# B&R Automation Studio project MOCS_AS
Automation Studio 4.12.5.95 SP

## Configuration GE3

CPU X20CP1686X, AutomationRuntime K4.93, Build 4.1.2, Vc V4.73.1

### Task classes (Cpu.sw)
```
Cyclic#4:
  IODiver <- IODefinitions.IODiver.prg
  CtrlLogic <- CtrlLogic.prg [disabled] (AdditionalIncludeDirectories=\Logical\MATLAB_includes\R2022b\, BuildOptions=-lm -DMODEL=MOCS_AS_Gen -DNUMST=1 -DNCSTATES=0 -DHAVESTDIO -DMODEL_HAS_DYNAMICALLY_LOADED_SFCNS=0 -DCLASSIC_INTERFACE=0 -DALLOCATIONFCN=0 -DTID01EQ=0 -DTERMFCN=1 -DONESTEPFCN=0 -DMAT_FILE=0 -DMULTI_INSTANCE_CODE=0 -DINTEGER_CODE=0 -DMT=0 )
Binaries: FWRules, udbdef, TCData, sysconf, asfw, User, iomap, arconfig, ashwd, Role, ashwac
Libraries: brsystem, asieccon, astime, runtime, sys_lib
```

### Hardware
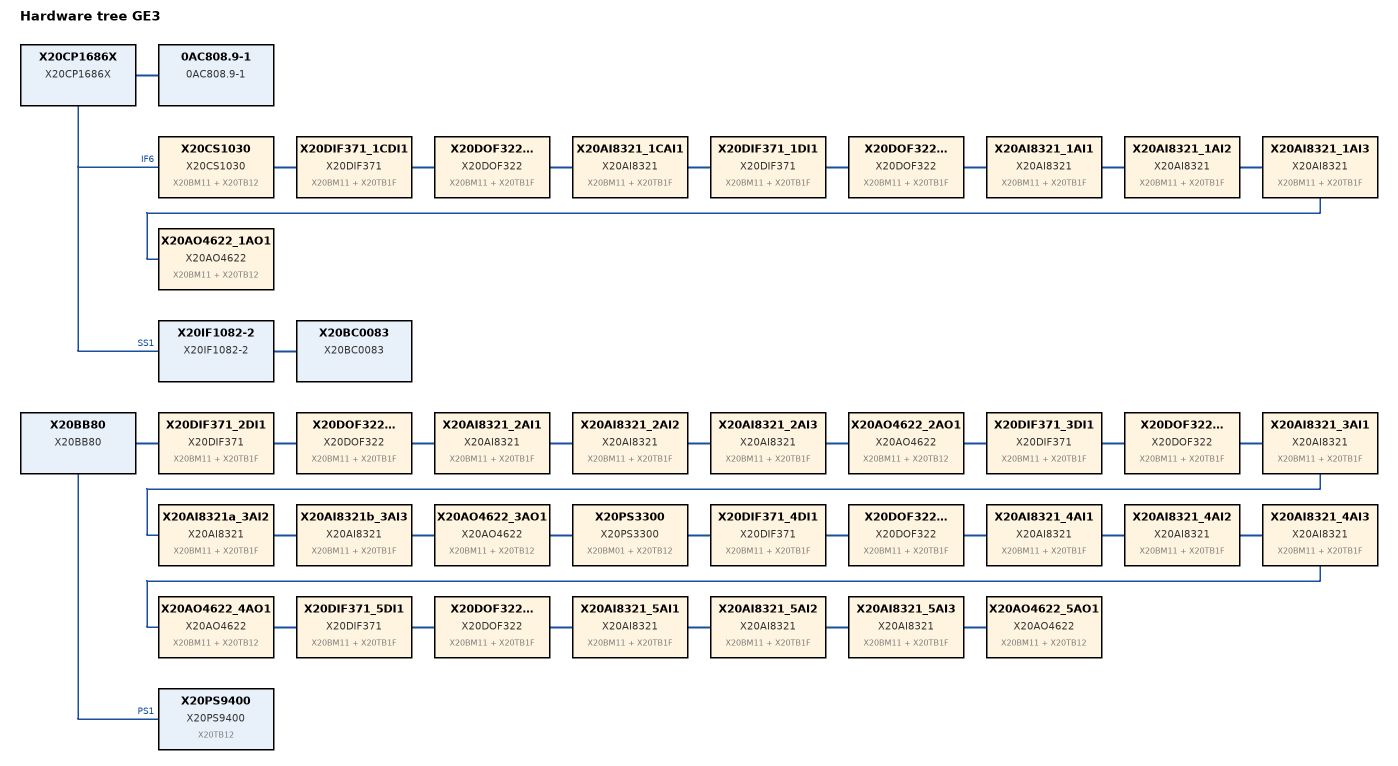
```
0AC808.9-1 : 0AC808.9-1 v1.0.0.0  [ETH1 -> X20CP1686X.IF2 [Cable Type=PowerlinkCable, Length=10, Version=1.0.0.3]]
X20AI8321_1AI1 : X20AI8321 v1.5.0.0  [SS1 -> X20TB1F5.SS; SL -> X20BM11f.SL1]
X20AI8321_1AI2 : X20AI8321 v1.5.0.0  [SS1 -> X20TB1F6.SS; SL -> X20BM11g.SL1]
X20AI8321_1AI3 : X20AI8321 v1.5.0.0  [SS1 -> X20TB1F7.SS; SL -> X20BM11h.SL1]
X20AI8321_1CAI1 : X20AI8321 v1.5.0.0  [SS1 -> X20TB1F2.SS; SL -> X20BM11c.SL1]
X20AI8321_2AI1 : X20AI8321 v1.5.0.0  [SS1 -> X20TB1F11.SS; SL -> X20BM11m.SL1]
X20AI8321_2AI2 : X20AI8321 v1.5.0.0  [SS1 -> X20TB1F12.SS; SL -> X20BM11n.SL1]
X20AI8321_2AI3 : X20AI8321 v1.5.0.0  [SS1 -> X20TB1F13.SS; SL -> X20BM11o.SL1]
X20AI8321_3AI1 : X20AI8321 v1.5.0.0  [SS1 -> X20TB1F15.SS; SL -> X20BM11r.SL1]
X20AI8321_4AI1 : X20AI8321 v1.5.0.0  [SS1 -> X20TB1F20.SS; SL -> X20BM11x.SL1]
X20AI8321_4AI2 : X20AI8321 v1.5.0.0  [SS1 -> X20TB1F21.SS; SL -> X20BM11y.SL1]
X20AI8321_4AI3 : X20AI8321 v1.5.0.0  [SS1 -> X20TB1F22.SS; SL -> X20BM11z.SL1]
X20AI8321_5AI1 : X20AI8321 v1.5.0.0  [SS1 -> X20TB1F25.SS; SL -> X20BM11ad.SL1]
X20AI8321_5AI2 : X20AI8321 v1.5.0.0  [SS1 -> X20TB1F26.SS; SL -> X20BM11ae.SL1]
X20AI8321_5AI3 : X20AI8321 v1.5.0.0  [SS1 -> X20TB1F27.SS; SL -> X20BM11af.SL1]
X20AI8321a_3AI2 : X20AI8321 v1.5.0.0  [SS1 -> X20TB1F16.SS; SL -> X20BM11s.SL1]
X20AI8321b_3AI3 : X20AI8321 v1.5.0.0  [SS1 -> X20TB1F17.SS; SL -> X20BM11t.SL1]
X20AO4622_1AO1 : X20AO4622 v1.4.1.0  [SS1 -> X20TB12a.SS; SL -> X20BM11i.SL1]
X20AO4622_2AO1 : X20AO4622 v1.4.1.0  [SS1 -> X20TB12c.SS; SL -> X20BM11l.SL1]
X20AO4622_3AO1 : X20AO4622 v1.4.1.0  [SS1 -> X20TB12d.SS; SL -> X20BM11u.SL1]
X20AO4622_4AO1 : X20AO4622 v1.4.1.0  [SS1 -> X20TB12e.SS; SL -> X20BM11aa.SL1]
X20AO4622_5AO1 : X20AO4622 v1.4.1.0  [SS1 -> X20TB12g.SS; SL -> X20BM11ag.SL1]
X20BB80 : X20BB80 v1.1.0.0
X20BC0083 : X20BC0083 v2.16.0.0  [PLK1 -> X20IF1082-2.IF1 (NodeNumber=1) [Cable Type=PowerlinkCable, Length=10, Version=1.0.0.3]; SL -> X20BB80.SL1]
X20BM01 : X20BM01 v2.2.0.0  [X2X1 -> X20BM11u.X2X2]
X20BM11 : X20BM11 v1.1.0.0  [X2X1 -> X20CP1686X.IF6]
X20BM11a : X20BM11 v1.1.0.0  [X2X1 -> X20BM11.X2X2]
X20BM11aa : X20BM11 v1.1.0.0  [X2X1 -> X20BM11z.X2X2]
X20BM11ab : X20BM11 v1.1.0.0  [X2X1 -> X20BM11aa.X2X2]
X20BM11ac : X20BM11 v1.1.0.0  [X2X1 -> X20BM11ab.X2X2]
X20BM11ad : X20BM11 v1.1.0.0  [X2X1 -> X20BM11ac.X2X2]
X20BM11ae : X20BM11 v1.1.0.0  [X2X1 -> X20BM11ad.X2X2]
X20BM11af : X20BM11 v1.1.0.0  [X2X1 -> X20BM11ae.X2X2]
X20BM11ag : X20BM11 v1.1.0.0  [X2X1 -> X20BM11af.X2X2]
X20BM11b : X20BM11 v1.1.0.0  [X2X1 -> X20BM11a.X2X2]
X20BM11c : X20BM11 v1.1.0.0  [X2X1 -> X20BM11b.X2X2]
X20BM11d : X20BM11 v1.1.0.0  [X2X1 -> X20BM11c.X2X2]
X20BM11e : X20BM11 v1.1.0.0  [X2X1 -> X20BM11d.X2X2]
X20BM11f : X20BM11 v1.1.0.0  [X2X1 -> X20BM11e.X2X2]
X20BM11g : X20BM11 v1.1.0.0  [X2X1 -> X20BM11f.X2X2]
X20BM11h : X20BM11 v1.1.0.0  [X2X1 -> X20BM11g.X2X2]
X20BM11i : X20BM11 v1.1.0.0  [X2X1 -> X20BM11h.X2X2]
X20BM11j : X20BM11 v1.1.0.0  [X2X1 -> X20BB80.IF1]
X20BM11k : X20BM11 v1.1.0.0  [X2X1 -> X20BM11j.X2X2]
X20BM11l : X20BM11 v1.1.0.0  [X2X1 -> X20BM11o.X2X2]
X20BM11m : X20BM11 v1.1.0.0  [X2X1 -> X20BM11k.X2X2]
X20BM11n : X20BM11 v1.1.0.0  [X2X1 -> X20BM11m.X2X2]
X20BM11o : X20BM11 v1.1.0.0  [X2X1 -> X20BM11n.X2X2]
X20BM11p : X20BM11 v1.1.0.0  [X2X1 -> X20BM11l.X2X2]
X20BM11q : X20BM11 v1.1.0.0  [X2X1 -> X20BM11p.X2X2]
X20BM11r : X20BM11 v1.1.0.0  [X2X1 -> X20BM11q.X2X2]
X20BM11s : X20BM11 v1.1.0.0  [X2X1 -> X20BM11r.X2X2]
X20BM11t : X20BM11 v1.1.0.0  [X2X1 -> X20BM11s.X2X2]
X20BM11u : X20BM11 v1.1.0.0  [X2X1 -> X20BM11t.X2X2]
X20BM11v : X20BM11 v1.1.0.0  [X2X1 -> X20BM01.X2X2]
X20BM11w : X20BM11 v1.1.0.0  [X2X1 -> X20BM11v.X2X2]
X20BM11x : X20BM11 v1.1.0.0  [X2X1 -> X20BM11w.X2X2]
X20BM11y : X20BM11 v1.1.0.0  [X2X1 -> X20BM11x.X2X2]
X20BM11z : X20BM11 v1.1.0.0  [X2X1 -> X20BM11y.X2X2]
X20CP1686X : X20CP1686X v1.6.2.0
  Connector IF2:
    ActivateDevice = 1
    HostName = multimocs
    Mode = Manual
    InternetAddress = 172.16.8.77
    SubnetMask = 255.255.255.0
  Connector IF3:
    EplHostName = multimocs
    HostName = multimocs
  ConfigurationID = MultiMOCS
  FileDevice1
  FileDeviceName1 = USER
  FileDevicePath1 = F:\
  FileDevice2
  FileDeviceName2 = USB_DEVICE
  FileDevicePath2 = /bd0
  FileDevice3
  FileDeviceName3 = ALARM_HISTROY
  FileDevicePath3 = F:\ALARM_HISTROY
  FileDevice4
  FileDeviceName4 = RECIPE
  FileDevicePath4 = F:\RECIPE
  FileDevice5
  FileDeviceName5 = AUDIT
  FileDevicePath5 = F:\AUDIT
  TimeZone = 325
  EthernetHostName = multimocs
  FtpUser1
  FtpUsername1 = hhi
  FtpUserPassword1 = NOQKJFEIpCMGTGhB1oqHL8VzUKYS3v77UCmMnhUHHNQ=
  FtpUserSalt1 = B7uzC8IW
  FTPAccessRight1 = 0
  ActivateOpcUa = 1
  OpcUaInformationModels_PV_Version = 1
X20CS1030 : X20CS1030 v1.8.0.0  [SS1 -> X20TB12.SS; SL -> X20BM11.SL1]
X20DIF371_1CDI1 : X20DIF371 v1.4.0.0  [SS1 -> X20TB1F.SS; SL -> X20BM11a.SL1]
X20DIF371_1DI1 : X20DIF371 v1.4.0.0  [SS1 -> X20TB1F3.SS; SL -> X20BM11d.SL1]
X20DIF371_2DI1 : X20DIF371 v1.4.0.0  [SS1 -> X20TB1F8.SS; SL -> X20BM11j.SL1]
X20DIF371_3DI1 : X20DIF371 v1.4.0.0  [SS1 -> X20TB1F10.SS; SL -> X20BM11p.SL1]
X20DIF371_4DI1 : X20DIF371 v1.4.0.0  [SS1 -> X20TB1F18.SS; SL -> X20BM11v.SL1]
X20DIF371_5DI1 : X20DIF371 v1.4.0.0  [SS1 -> X20TB1F23.SS; SL -> X20BM11ab.SL1]
X20DOF322_1CDO1 : X20DOF322 v1.5.0.0  [SS1 -> X20TB1F1.SS; SL -> X20BM11b.SL1]
X20DOF322_1DO1 : X20DOF322 v1.5.0.0  [SS1 -> X20TB1F4.SS; SL -> X20BM11e.SL1]
X20DOF322_2DO1 : X20DOF322 v1.5.0.0  [SS1 -> X20TB1F9.SS; SL -> X20BM11k.SL1]
X20DOF322_3DO1 : X20DOF322 v1.5.0.0  [SS1 -> X20TB1F14.SS; SL -> X20BM11q.SL1]
X20DOF322_4DO1 : X20DOF322 v1.5.0.0  [SS1 -> X20TB1F19.SS; SL -> X20BM11w.SL1]
X20DOF322_5DO1 : X20DOF322 v1.5.0.0  [SS1 -> X20TB1F24.SS; SL -> X20BM11ac.SL1]
X20IF1082-2 : X20IF1082-2 v1.15.0.0  [SS -> X20CP1686X.SS1]
  Connector IF1:
    EplHostName = multimocs
    EplNatSubnet = 192.168.102.0
    HostName = multimocs
X20PS3300 : X20PS3300 v1.4.0.0  [SS1 -> X20TB12f.SS; SL -> X20BM01.SL1]
X20PS9400 : X20PS9400 v1.8.0.0  [SS1 -> X20TB12b.SS; PS -> X20BB80.PS1]
X20TB12 : X20TB12 v1.0.0.0
X20TB12a : X20TB12 v1.0.0.0
X20TB12b : X20TB12 v1.0.0.0
X20TB12c : X20TB12 v1.0.0.0
X20TB12d : X20TB12 v1.0.0.0
X20TB12e : X20TB12 v1.0.0.0
X20TB12f : X20TB12 v1.0.0.0
X20TB12g : X20TB12 v1.0.0.0
X20TB1F : X20TB1F v1.0.0.0
X20TB1F1 : X20TB1F v1.0.0.0
X20TB1F10 : X20TB1F v1.0.0.0
X20TB1F11 : X20TB1F v1.0.0.0
X20TB1F12 : X20TB1F v1.0.0.0
X20TB1F13 : X20TB1F v1.0.0.0
X20TB1F14 : X20TB1F v1.0.0.0
X20TB1F15 : X20TB1F v1.0.0.0
X20TB1F16 : X20TB1F v1.0.0.0
X20TB1F17 : X20TB1F v1.0.0.0
X20TB1F18 : X20TB1F v1.0.0.0
X20TB1F19 : X20TB1F v1.0.0.0
X20TB1F2 : X20TB1F v1.0.0.0
X20TB1F20 : X20TB1F v1.0.0.0
X20TB1F21 : X20TB1F v1.0.0.0
X20TB1F22 : X20TB1F v1.0.0.0
X20TB1F23 : X20TB1F v1.0.0.0
X20TB1F24 : X20TB1F v1.0.0.0
X20TB1F25 : X20TB1F v1.0.0.0
X20TB1F26 : X20TB1F v1.0.0.0
X20TB1F27 : X20TB1F v1.0.0.0
X20TB1F3 : X20TB1F v1.0.0.0
X20TB1F4 : X20TB1F v1.0.0.0
X20TB1F5 : X20TB1F v1.0.0.0
X20TB1F6 : X20TB1F v1.0.0.0
X20TB1F7 : X20TB1F v1.0.0.0
X20TB1F8 : X20TB1F v1.0.0.0
X20TB1F9 : X20TB1F v1.0.0.0
```

## Configuration TestConfig

CPU X20CP1686X, AutomationRuntime K4.93, Build 4.1.2, Vc V4.73.1

### Hardware
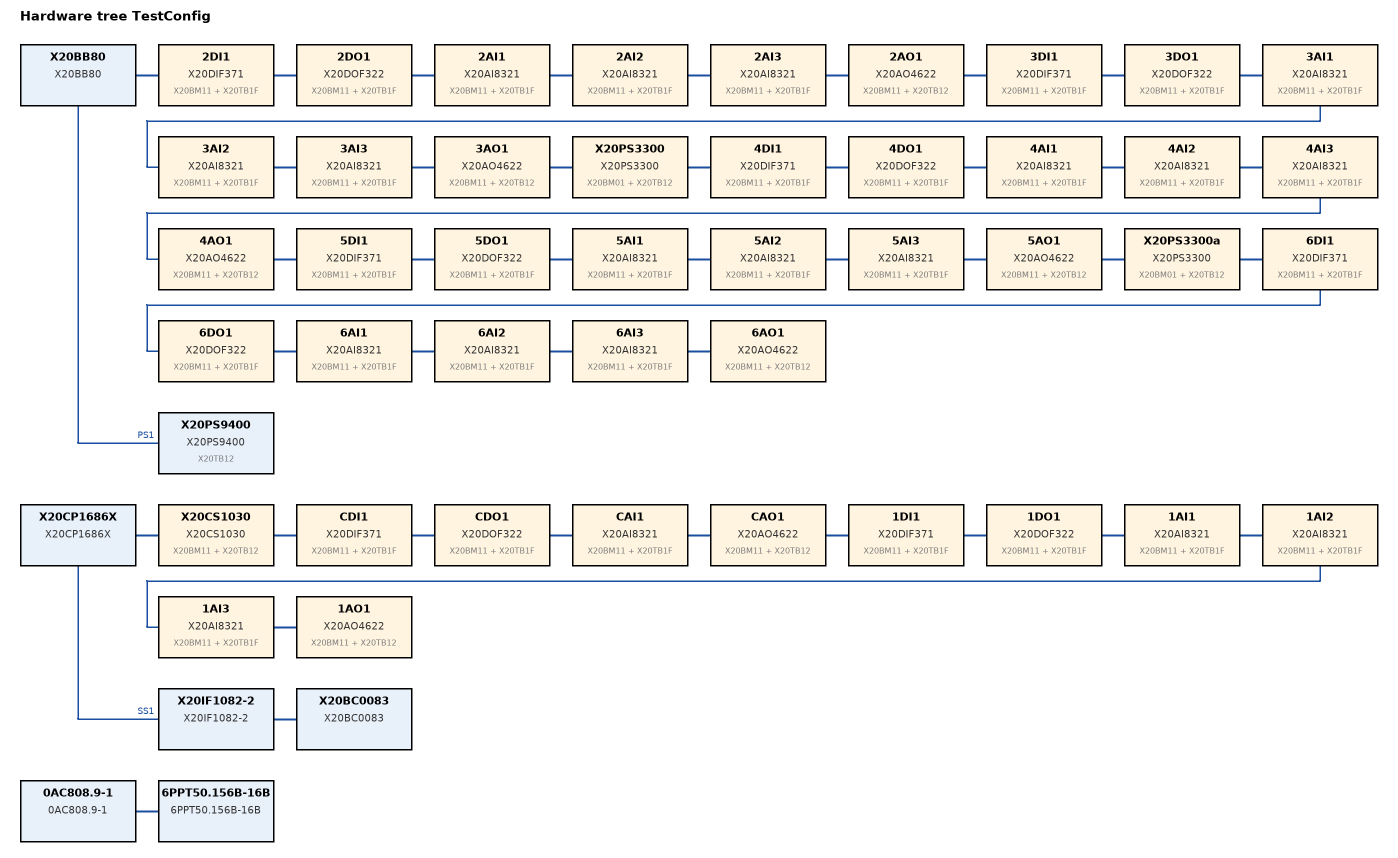
```
0AC808.9-1 : 0AC808.9-1 v1.0.0.0  [ETH1 -> 6PPT50.156B-16B.ETH2 [Cable Type=PowerlinkCable, Length=10, Version=1.0.0.3]; ETH5 -> X20CP1686X.IF2 [Cable Type=PowerlinkCable, Length=10, Version=1.0.0.3]]
1AI1 : X20AI8321 v1.5.0.0  [SS1 -> X20TB1F5.SS; SL -> X20BM11g.SL1]
1AI2 : X20AI8321 v1.5.0.0  [SS1 -> X20TB1F6.SS; SL -> X20BM11i.SL1]
1AI3 : X20AI8321 v1.5.0.0  [SS1 -> X20TB1F7.SS; SL -> X20BM11j.SL1]
1AO1 : X20AO4622 v1.4.1.0  [SS1 -> X20TB12b.SS; SL -> X20BM11h.SL1]
1DI1 : X20DIF371 v1.4.0.0  [SS1 -> X20TB1F3.SS; SL -> X20BM11e.SL1]
1DO1 : X20DOF322 v1.5.0.0  [SS1 -> X20TB1F4.SS; SL -> X20BM11f.SL1]
2AI1 : X20AI8321 v1.5.0.0  [SS1 -> X20TB1F9.SS; SL -> X20BM11l.SL1]
2AI2 : X20AI8321 v1.5.0.0  [SS1 -> X20TB1F10.SS; SL -> X20BM11m.SL1]
2AI3 : X20AI8321 v1.5.0.0  [SS1 -> X20TB1F11.SS; SL -> X20BM11n.SL1]
2AO1 : X20AO4622 v1.4.1.0  [SS1 -> X20TB12d.SS; SL -> X20BM11o.SL1]
2DI1 : X20DIF371 v1.4.0.0  [SS1 -> X20TB1F12.SS; SL -> X20BM11p.SL1]
2DO1 : X20DOF322 v1.5.0.0  [SS1 -> X20TB1F8.SS; SL -> X20BM11k.SL1]
3AI1 : X20AI8321 v1.5.0.0  [SS1 -> X20TB1F14.SS; SL -> X20BM11r.SL1]
3AI2 : X20AI8321 v1.5.0.0  [SS1 -> X20TB1F15.SS; SL -> X20BM11s.SL1]
3AI3 : X20AI8321 v1.5.0.0  [SS1 -> X20TB1F16.SS; SL -> X20BM11t.SL1]
3AO1 : X20AO4622 v1.4.1.0  [SS1 -> X20TB12e.SS; SL -> X20BM11u.SL1]
3DI1 : X20DIF371 v1.4.0.0  [SS1 -> X20TB1F17.SS; SL -> X20BM11v.SL1]
3DO1 : X20DOF322 v1.5.0.0  [SS1 -> X20TB1F13.SS; SL -> X20BM11q.SL1]
4AI1 : X20AI8321 v1.5.0.0  [SS1 -> X20TB1F30.SS; SL -> X20BM11ak.SL1]
4AI2 : X20AI8321 v1.5.0.0  [SS1 -> X20TB1F31.SS; SL -> X20BM11al.SL1]
4AI3 : X20AI8321 v1.5.0.0  [SS1 -> X20TB1F32.SS; SL -> X20BM11am.SL1]
4AO1 : X20AO4622 v1.4.1.0  [SS1 -> X20TB12j.SS; SL -> X20BM11an.SL1]
4DI1 : X20DIF371 v1.4.0.0  [SS1 -> X20TB1F28.SS; SL -> X20BM11ai.SL1]
4DO1 : X20DOF322 v1.5.0.0  [SS1 -> X20TB1F29.SS; SL -> X20BM11aj.SL1]
5AI1 : X20AI8321 v1.5.0.0  [SS1 -> X20TB1F35.SS; SL -> X20BM11aq.SL1]
5AI2 : X20AI8321 v1.5.0.0  [SS1 -> X20TB1F36.SS; SL -> X20BM11ar.SL1]
5AI3 : X20AI8321 v1.5.0.0  [SS1 -> X20TB1F37.SS; SL -> X20BM11as.SL1]
5AO1 : X20AO4622 v1.4.1.0  [SS1 -> X20TB12k.SS; SL -> X20BM11at.SL1]
5DI1 : X20DIF371 v1.4.0.0  [SS1 -> X20TB1F33.SS; SL -> X20BM11ao.SL1]
5DO1 : X20DOF322 v1.5.0.0  [SS1 -> X20TB1F34.SS; SL -> X20BM11ap.SL1]
6AI1 : X20AI8321 v1.5.0.0  [SS1 -> X20TB1F40.SS; SL -> X20BM11aw.SL1]
6AI2 : X20AI8321 v1.5.0.0  [SS1 -> X20TB1F41.SS; SL -> X20BM11ax.SL1]
6AI3 : X20AI8321 v1.5.0.0  [SS1 -> X20TB1F42.SS; SL -> X20BM11ay.SL1]
6AO1 : X20AO4622 v1.4.1.0  [SS1 -> X20TB12m.SS; SL -> X20BM11az.SL1]
6DI1 : X20DIF371 v1.4.0.0  [SS1 -> X20TB1F38.SS; SL -> X20BM11au.SL1]
6DO1 : X20DOF322 v1.5.0.0  [SS1 -> X20TB1F39.SS; SL -> X20BM11av.SL1]
6PPT50.156B-16B : 6PPT50.156B-16B v1.3.8.0  [ETH2 -> 0AC808.9-1.ETH1 [Cable Type=PowerlinkCable, Length=10, Version=1.0.0.3]]
  Terminal = true
  PasswordVNC = 
  PasswordCIFS = 
  PasswordService = 
CAI1 : X20AI8321 v1.5.0.0  [SS1 -> X20TB1F2.SS; SL -> X20BM11c.SL1]
CAO1 : X20AO4622 v1.4.1.0  [SS1 -> X20TB12a.SS; SL -> X20BM11d.SL1]
CDI1 : X20DIF371 v1.4.0.0  [SS1 -> X20TB1F.SS; SL -> X20BM11a.SL1]
CDO1 : X20DOF322 v1.5.0.0  [SS1 -> X20TB1F1.SS; SL -> X20BM11b.SL1]
X20BB80 : X20BB80 v1.1.0.0
X20BC0083 : X20BC0083 v2.14.0.0  [PLK1 -> X20IF1082-2.IF1 (NodeNumber=1) [Cable Type=PowerlinkCable, Length=10, Version=1.0.0.3]; SL -> X20BB80.SL1]
X20BM01 : X20BM01 v2.2.0.0  [X2X1 -> X20BM11u.X2X2]
X20BM01a : X20BM01 v2.2.0.0  [X2X1 -> X20BM11at.X2X2]
X20BM11 : X20BM11 v1.1.0.0  [X2X1 -> X20CP1686X.IF6]
X20BM11a : X20BM11 v1.1.0.0  [X2X1 -> X20BM11.X2X2]
X20BM11ai : X20BM11 v1.1.0.0  [X2X1 -> X20BM01.X2X2]
X20BM11aj : X20BM11 v1.1.0.0  [X2X1 -> X20BM11ai.X2X2]
X20BM11ak : X20BM11 v1.1.0.0  [X2X1 -> X20BM11aj.X2X2]
X20BM11al : X20BM11 v1.1.0.0  [X2X1 -> X20BM11ak.X2X2]
X20BM11am : X20BM11 v1.1.0.0  [X2X1 -> X20BM11al.X2X2]
X20BM11an : X20BM11 v1.1.0.0  [X2X1 -> X20BM11am.X2X2]
X20BM11ao : X20BM11 v1.1.0.0  [X2X1 -> X20BM11an.X2X2]
X20BM11ap : X20BM11 v1.1.0.0  [X2X1 -> X20BM11ao.X2X2]
X20BM11aq : X20BM11 v1.1.0.0  [X2X1 -> X20BM11ap.X2X2]
X20BM11ar : X20BM11 v1.1.0.0  [X2X1 -> X20BM11aq.X2X2]
X20BM11as : X20BM11 v1.1.0.0  [X2X1 -> X20BM11ar.X2X2]
X20BM11at : X20BM11 v1.1.0.0  [X2X1 -> X20BM11as.X2X2]
X20BM11au : X20BM11 v1.1.0.0  [X2X1 -> X20BM01a.X2X2]
X20BM11av : X20BM11 v1.1.0.0  [X2X1 -> X20BM11au.X2X2]
X20BM11aw : X20BM11 v1.1.0.0  [X2X1 -> X20BM11av.X2X2]
X20BM11ax : X20BM11 v1.1.0.0  [X2X1 -> X20BM11aw.X2X2]
X20BM11ay : X20BM11 v1.1.0.0  [X2X1 -> X20BM11ax.X2X2]
X20BM11az : X20BM11 v1.1.0.0  [X2X1 -> X20BM11ay.X2X2]
X20BM11b : X20BM11 v1.1.0.0  [X2X1 -> X20BM11a.X2X2]
X20BM11c : X20BM11 v1.1.0.0  [X2X1 -> X20BM11b.X2X2]
X20BM11d : X20BM11 v1.1.0.0  [X2X1 -> X20BM11c.X2X2]
X20BM11e : X20BM11 v1.1.0.0  [X2X1 -> X20BM11d.X2X2]
X20BM11f : X20BM11 v1.1.0.0  [X2X1 -> X20BM11e.X2X2]
X20BM11g : X20BM11 v1.1.0.0  [X2X1 -> X20BM11f.X2X2]
X20BM11h : X20BM11 v1.1.0.0  [X2X1 -> X20BM11j.X2X2]
X20BM11i : X20BM11 v1.1.0.0  [X2X1 -> X20BM11g.X2X2]
X20BM11j : X20BM11 v1.1.0.0  [X2X1 -> X20BM11i.X2X2]
X20BM11k : X20BM11 v1.1.0.0  [X2X1 -> X20BM11p.X2X2]
X20BM11l : X20BM11 v1.1.0.0  [X2X1 -> X20BM11k.X2X2]
X20BM11m : X20BM11 v1.1.0.0  [X2X1 -> X20BM11l.X2X2]
X20BM11n : X20BM11 v1.1.0.0  [X2X1 -> X20BM11m.X2X2]
X20BM11o : X20BM11 v1.1.0.0  [X2X1 -> X20BM11n.X2X2]
X20BM11p : X20BM11 v1.1.0.0  [X2X1 -> X20BB80.IF1]
X20BM11q : X20BM11 v1.1.0.0  [X2X1 -> X20BM11v.X2X2]
X20BM11r : X20BM11 v1.1.0.0  [X2X1 -> X20BM11q.X2X2]
X20BM11s : X20BM11 v1.1.0.0  [X2X1 -> X20BM11r.X2X2]
X20BM11t : X20BM11 v1.1.0.0  [X2X1 -> X20BM11s.X2X2]
X20BM11u : X20BM11 v1.1.0.0  [X2X1 -> X20BM11t.X2X2]
X20BM11v : X20BM11 v1.1.0.0  [X2X1 -> X20BM11o.X2X2]
X20CP1686X : X20CP1686X v1.6.2.0
  Connector IF2:
    ActivateDevice = 1
    HostName = multimocs
    Mode = Manual
    InternetAddress = 172.16.8.77
    SubnetMask = 255.255.255.0
  Connector IF3:
    EplHostName = multimocs
    HostName = multimocs
  ConfigurationID = MultiMOCS
  FileDevice1
  FileDeviceName1 = USER
  FileDevicePath1 = F:\
  FileDevice2
  FileDeviceName2 = USB_DEVICE
  FileDevicePath2 = /bd0
  FileDevice3
  FileDeviceName3 = ALARM_HISTROY
  FileDevicePath3 = F:\ALARM_HISTROY
  FileDevice4
  FileDeviceName4 = RECIPE
  FileDevicePath4 = F:\RECIPE
  FileDevice5
  FileDeviceName5 = AUDIT
  FileDevicePath5 = F:\AUDIT
  TimeZone = 325
  EthernetHostName = multimocs
  FtpUser1
  FtpUsername1 = hhi
  FtpUserPassword1 = NOQKJFEIpCMGTGhB1oqHL8VzUKYS3v77UCmMnhUHHNQ=
  FtpUserSalt1 = B7uzC8IW
  FTPAccessRight1 = 0
  ActivateOpcUa = 1
  OpcUaInformationModels_PV_Version = 1
X20CS1030 : X20CS1030 v1.8.0.0  [SS1 -> X20TB12.SS; SL -> X20BM11.SL1]
X20IF1082-2 : X20IF1082-2 v1.15.0.0  [SS -> X20CP1686X.SS1]
  Connector IF1:
    EplNatSubnet = 192.168.102.0
X20PS3300 : X20PS3300 v1.4.0.0  [SS1 -> X20TB12i.SS; SL -> X20BM01.SL1]
X20PS3300a : X20PS3300 v1.4.0.0  [SS1 -> X20TB12l.SS; SL -> X20BM01a.SL1]
X20PS9400 : X20PS9400 v1.8.0.0  [SS1 -> X20TB12c.SS; PS -> X20BB80.PS1]
X20TB12 : X20TB12 v1.0.0.0
X20TB12a : X20TB12 v1.0.0.0
X20TB12b : X20TB12 v1.0.0.0
X20TB12c : X20TB12 v1.0.0.0
X20TB12d : X20TB12 v1.0.0.0
X20TB12e : X20TB12 v1.0.0.0
X20TB12i : X20TB12 v1.0.0.0
X20TB12j : X20TB12 v1.0.0.0
X20TB12k : X20TB12 v1.0.0.0
X20TB12l : X20TB12 v1.0.0.0
X20TB12m : X20TB12 v1.0.0.0
X20TB1F : X20TB1F v1.0.0.0
X20TB1F1 : X20TB1F v1.0.0.0
X20TB1F10 : X20TB1F v1.0.0.0
X20TB1F11 : X20TB1F v1.0.0.0
X20TB1F12 : X20TB1F v1.0.0.0
X20TB1F13 : X20TB1F v1.0.0.0
X20TB1F14 : X20TB1F v1.0.0.0
X20TB1F15 : X20TB1F v1.0.0.0
X20TB1F16 : X20TB1F v1.0.0.0
X20TB1F17 : X20TB1F v1.0.0.0
X20TB1F2 : X20TB1F v1.0.0.0
X20TB1F28 : X20TB1F v1.0.0.0
X20TB1F29 : X20TB1F v1.0.0.0
X20TB1F3 : X20TB1F v1.0.0.0
X20TB1F30 : X20TB1F v1.0.0.0
X20TB1F31 : X20TB1F v1.0.0.0
X20TB1F32 : X20TB1F v1.0.0.0
X20TB1F33 : X20TB1F v1.0.0.0
X20TB1F34 : X20TB1F v1.0.0.0
X20TB1F35 : X20TB1F v1.0.0.0
X20TB1F36 : X20TB1F v1.0.0.0
X20TB1F37 : X20TB1F v1.0.0.0
X20TB1F38 : X20TB1F v1.0.0.0
X20TB1F39 : X20TB1F v1.0.0.0
X20TB1F4 : X20TB1F v1.0.0.0
X20TB1F40 : X20TB1F v1.0.0.0
X20TB1F41 : X20TB1F v1.0.0.0
X20TB1F42 : X20TB1F v1.0.0.0
X20TB1F5 : X20TB1F v1.0.0.0
X20TB1F6 : X20TB1F v1.0.0.0
X20TB1F7 : X20TB1F v1.0.0.0
X20TB1F8 : X20TB1F v1.0.0.0
X20TB1F9 : X20TB1F v1.0.0.0
```

## Logical view

Binary libraries used (declarations not repeated): operator, runtime, astime, AsIecCon, brsystem, sys_lib

### Global.var - Global variables
```iecst
VAR
	OpcUA_mon : ARRAY[0..20] OF INT := [0,1,2,3,4,5,6,7,8,9,10,11,12,13,14,15,16,17,18,19,20];
	OpcUA_cmd : ARRAY[0..10] OF INT;
	OpcUA_modifier : ARRAY[0..70] OF USINT;
	OpcUA_set_1 : ARRAY[0..10] OF INT;
	IF_MON : ARRAY[0..199] OF REAL;
	IF_MON1 : ARRAY[0..99] OF REAL;
	IF_MON2 : ARRAY[0..99] OF REAL;
	IF_MON3 : ARRAY[0..99] OF REAL;
	IF_MON4 : ARRAY[0..99] OF REAL;
	IF_MON5 : ARRAY[0..99] OF REAL;
	IF_MON6 : ARRAY[0..99] OF REAL;
	IF_MON7 : ARRAY[0..99] OF REAL;
	IF_MON8 : ARRAY[0..99] OF REAL;
END_VAR
```

### RcpTypes.typ
```iecst
(*---Category1---*)

TYPE
	Para_typ : 	STRUCT  (*Comm[0..199], Indiv[0..99]*8*)
		Common : ParaCommon_typ;
		No1 : ParaIndiv_typ;
		No2 : ParaIndiv_typ;
		No3 : ParaIndiv_typ;
		No4 : ParaIndiv_typ;
		No5 : ParaIndiv_typ;
		No6 : ParaIndiv_typ;
		No7 : ParaIndiv_typ;
		No8 : ParaIndiv_typ;
	END_STRUCT;
END_TYPE

(*---Category2---*)

TYPE
	ParaCommon_typ : 	STRUCT  (*Comm[0..199]*)
		System : System_typ; (*Comm[0..49]*)
		StateFlag : StateFlag_typ; (*Comm[50..99]: 50*)
		Main : Main_typ; (*Comm[100..149]: 50*)
		FODS : FODS_typ; (*Comm[150..179]*)
		CommonReservedCat2 : CommonReservedCat2_typ; (*Comm[180..199]*)
	END_STRUCT;
	ParaIndiv_typ : 	STRUCT  (*Indiv[0..99]*)
		FODSFeedforward : FODSFeedforward_typ; (*[0..49]: 50*)
		FODSFeedback : FODSFeedback_typ; (*[50..74]: 25*)
		IndivReservedCat2 : IndivReservedCat2_typ; (*[75..99]*)
	END_STRUCT;
END_TYPE

(*---Category3---*)

TYPE
	System_typ : 	STRUCT  (*Comm[0..49]: 50*)
		SystemType : SystemType_typ;
		CommSetting : CommSetting_typ;
		SystemReserved : SystemReserved_typ;
	END_STRUCT;
	StateFlag_typ : 	STRUCT  (*Comm[50..99]: 50*)
		MSSNormalFlag : MSSNormalFlag_typ; (*[50..54]: 5*)
		LoadChangeFlag : LoadChangeFlag_typ; (*[55:59]: 5*)
		SystemWarmedUpFlag : SystemWarmedUpFlag_typ; (*[60..64]: 5*)
		TMBFlag : TMBFlag_typ; (*[65..99]: 35*)
		FlagReserved : FlagReserved_typ; (*[65..99]: 35*)
	END_STRUCT;
	Main_typ : 	STRUCT  (*Comm[100..149]: 50*)
		Init : Init_typ;
		Sealing : Sealing_typ;
		Engage : Engage_typ;
		Active : Active_typ;
		TMB : TMB_typ;
		Disengage : Disengage_typ;
		Airventing : Airventing_typ;
		MOCSshutdown : MOCSshutdown_typ;
		Valveshutdown : Valveshutdown_typ;
	END_STRUCT;
	FODS_typ : 	STRUCT  (*Comm[150..179]: 30*)
		FODSInitReady : FODSInitReady_typ;
		FODSCooling : FODSCooling_typ;
		FODSDosing : FODSDosing_typ;
		FODSFlushing : FODSFlushing_typ;
	END_STRUCT;
	CommonReservedCat2_typ : 	STRUCT
		CommonReservedCat3 : CommonReservedCat3_typ;
	END_STRUCT;
	FODSFeedforward_typ : 	STRUCT  (*Indiv[0..49]: 50*)
		FFpara : FFpara_typ;
		EngineLoad : EngineLoad_typ;
		ExhFlowrate : ExhFlowrate_typ;
		HUInletRefTemp : HUInletRefTemp_typ;
		CorrectionFactor : CorrectionFactor_typ;
	END_STRUCT;
	FODSFeedback_typ : 	STRUCT  (*Indiv[50..74]: 25*)
		MOCSTempPgain : MOCSTempPgain_typ;
		APIDgain : APIDgain_typ;
	END_STRUCT;
	IndivReservedCat2_typ : 	STRUCT  (*Indiv[75..99]: 25*)
		IndivReservedCat3 : IndivReservedCat3_typ;
	END_STRUCT;
END_TYPE

(*---Category4---*)

TYPE
	SystemType_typ : 	STRUCT  (*Comm[0..9]: 10*)
		MOCSType : REAL; (*[0]*)
		NumofGE : REAL; (*[1]*)
		HeatingSystem : REAL; (*[2]*)
		FOSuppUnit : REAL; (*[4]*)
		SystemTypeReserved4 : REAL;
		SystemTypeReserved5 : REAL;
		SystemTypeReserved6 : REAL;
		SystemTypeReserved7 : REAL;
		SystemTypeReserved8 : REAL;
		SystemTypeReserved9 : REAL;
	END_STRUCT;
	CommSetting_typ : 	STRUCT  (*Comm[10..14]: 5*)
		ValveStatusCriteria : REAL;
		FOPumpChangeOverTime : REAL;
		FOPumpChangeOverDelay : REAL;
		CommSettingReserved3 : REAL;
		CommSettingReserved4 : REAL;
	END_STRUCT;
	SystemReserved_typ : 	STRUCT  (*Comm[15..49]: 35*)
		SystemReserved15 : REAL;
		SystemReserved16 : REAL;
		SystemReserved17 : REAL;
		SystemReserved18 : REAL;
		SystemReserved19 : REAL;
		SystemReserved20 : REAL;
		SystemReserved21 : REAL;
		SystemReserved22 : REAL;
		SystemReserved23 : REAL;
		SystemReserved24 : REAL;
		SystemReserved25 : REAL;
		SystemReserved26 : REAL;
		SystemReserved27 : REAL;
		SystemReserved28 : REAL;
		SystemReserved29 : REAL;
		SystemReserved30 : REAL;
		SystemReserved31 : REAL;
		SystemReserved32 : REAL;
		SystemReserved33 : REAL;
		SystemReserved34 : REAL;
		SystemReserved35 : REAL;
		SystemReserved36 : REAL;
		SystemReserved37 : REAL;
		SystemReserved38 : REAL;
		SystemReserved39 : REAL;
		SystemReserved40 : REAL;
		SystemReserved41 : REAL;
		SystemReserved42 : REAL;
		SystemReserved43 : REAL;
		SystemReserved44 : REAL;
		SystemReserved45 : REAL;
		SystemReserved46 : REAL;
		SystemReserved47 : REAL;
		SystemReserved48 : REAL;
		SystemReserved49 : REAL;
	END_STRUCT;
	MSSNormalFlag_typ : 	STRUCT  (*Comm[50..54]: 5*)
		MOCSMinEngineLoad : REAL;
		MOCSReadyEngineLoad : REAL;
		MSSNormalFallingHysteresis : REAL;
		MSSNormalFallingDelay : REAL;
		MSSFlagReserved4 : REAL;
	END_STRUCT;
	LoadChangeFlag_typ : 	STRUCT  (*Comm[55..59]: 5*)
		MovAvgPeriod : REAL;
		ComparePoint : REAL;
		LoadChangeThreshold : REAL;
		LoadChangeFlagReserved3 : REAL;
		LoadChangeFlagReserved4 : REAL;
	END_STRUCT;
	SystemWarmedUpFlag_typ : 	STRUCT  (*Comm[60..64]: 5*)
		WarmUpDTemp : REAL;
		WarmUpITemp : REAL;
		WarmUpChITemp : REAL;
		WarmUpChMTemp : REAL;
		WarmUpChOTemp : REAL;
	END_STRUCT;
	TMBFlag_typ : 	STRUCT  (*Comm[65..69]: 5*)
		TMBFlagFallingDelay : REAL;
		TMBFlagReserved1 : REAL;
		TMBFlagReserved2 : REAL;
		TMBFlagReserved3 : REAL;
		TMBFlagReserved4 : REAL;
	END_STRUCT;
	FlagReserved_typ : 	STRUCT  (*Comm[70..99]: 30*)
		FlagReserved20 : REAL;
		FlagReserved21 : REAL;
		FlagReserved22 : REAL;
		FlagReserved23 : REAL;
		FlagReserved24 : REAL;
		FlagReserved25 : REAL;
		FlagReserved26 : REAL;
		FlagReserved27 : REAL;
		FlagReserved28 : REAL;
		FlagReserved29 : REAL;
		FlagReserved30 : REAL;
		FlagReserved31 : REAL;
		FlagReserved32 : REAL;
		FlagReserved33 : REAL;
		FlagReserved34 : REAL;
		FlagReserved35 : REAL;
		FlagReserved36 : REAL;
		FlagReserved37 : REAL;
		FlagReserved38 : REAL;
		FlagReserved39 : REAL;
		FlagReserved40 : REAL;
		FlagReserved41 : REAL;
		FlagReserved42 : REAL;
		FlagReserved43 : REAL;
		FlagReserved44 : REAL;
		FlagReserved45 : REAL;
		FlagReserved46 : REAL;
		FlagReserved47 : REAL;
		FlagReserved48 : REAL;
		FlagReserved49 : REAL;
	END_STRUCT;
	Init_typ : 	STRUCT  (*Comm[100..104]: 5*)
		InitReserved0 : REAL;
		InitReserved1 : REAL;
		InitReserved2 : REAL;
		InitReserved3 : REAL;
		InitReserved4 : REAL;
	END_STRUCT;
	Sealing_typ : 	STRUCT  (*Comm[105..114]: 10*)
		VSSolValveOpenDP : REAL;
		VSSolValveCloseDP : REAL;
		RTVOpenDP : REAL;
		RTVCloseDP : REAL;
		SealRTVSetpoint : REAL;
		VSSolValveOpenDuration : REAL;
		VSSolValveCloseDuration : REAL;
		SealingReserved7 : REAL;
		SealingReserved8 : REAL;
		SealingReserved9 : REAL;
	END_STRUCT;
	Engage_typ : 	STRUCT  (*Comm[115..119]: 5*)
		EnRTVSlope : REAL;
		EngageReserved1 : REAL;
		EngageReserved2 : REAL;
		EngageReserved3 : REAL;
		EngageReserved4 : REAL;
	END_STRUCT;
	Active_typ : 	STRUCT  (*Comm[120..124]: 5*)
		HUTargetTemp : REAL;
		HUActiveTemp : REAL;
		HUInactiveOffsetTemp : REAL;
		ActiveReserved3 : REAL;
		ActiveReserved4 : REAL;
	END_STRUCT;
	TMB_typ : 	STRUCT  (*Comm[125..129]: 5*)
		TMBBypassMinDuration : REAL;
		TMBTimeoutThreshold : REAL;
		TMBReserved2 : REAL;
		TMBReserved3 : REAL;
		TMBReserved4 : REAL;
	END_STRUCT;
	Disengage_typ : 	STRUCT  (*Comm[130..134]: 5*)
		DisenRTVSlope : REAL;
		DisengageReserved1 : REAL;
		DisengageReserved2 : REAL;
		DisengageReserved3 : REAL;
		DisengageReserved4 : REAL;
	END_STRUCT;
	Airventing_typ : 	STRUCT  (*Comm[135..139]: 5*)
		VentRTVSetpoint : REAL;
		VentDuration : REAL;
		AirVentingReserved2 : REAL;
		AirVentingReserved3 : REAL;
		AirVentingReserved4 : REAL;
	END_STRUCT;
	MOCSshutdown_typ : 	STRUCT  (*Comm[140..144]: 5*)
		MOCSShutdownReserved0 : REAL;
		MOCSShutdownReserved1 : REAL;
		MOCSShutdownReserved2 : REAL;
		MOCSShutdownReserved3 : REAL;
		MOCSShutdownReserved4 : REAL;
	END_STRUCT;
	Valveshutdown_typ : 	STRUCT  (*Comm[145..149]: 5*)
		ValveShutdownReserved0 : REAL;
		ValveShutdownReserved1 : REAL;
		ValveShutdownReserved2 : REAL;
		ValveShutdownReserved3 : REAL;
		ValveShutdownReserved4 : REAL;
	END_STRUCT;
	FODSInitReady_typ : 	STRUCT  (*Comm[150..154]: 5*)
		FODSInitReserved0 : REAL;
		FODSInitReserved1 : REAL;
		FODSInitReserved2 : REAL;
		FODSInitReserved3 : REAL;
		FODSInitReserved4 : REAL;
	END_STRUCT;
	FODSCooling_typ : 	STRUCT  (*Comm[155..159]: 5*)
		FOCoolDuration : REAL;
		FODSCoolingReserved1 : REAL;
		FODSCoolingReserved2 : REAL;
		FODSCoolingReserved3 : REAL;
		FODSCoolingReserved4 : REAL;
	END_STRUCT;
	FODSDosing_typ : 	STRUCT  (*Comm[160..174]: 15*)
		PumpChangeOverTime : REAL;
		SolVVDelay : REAL;
		LowRefQFOTimeout : REAL;
		QFOLowLimitTimeout : REAL;
		SFFlowrateThHigh : REAL;
		SFFlowrateThLow : REAL;
		QFOHighLimitGain : REAL;
		QFOHighLimitMin : REAL;
		QFOLowLimitValue : REAL;
		FOCValHighLimitValue : REAL;
		FOCValLowLimitValue : REAL;
		FODSDosingReserved11 : REAL;
		FODSDosingReserved12 : REAL;
		FODSDosingReserved13 : REAL;
		FODSDosingReserved14 : REAL;
	END_STRUCT;
	FODSFlushing_typ : 	STRUCT  (*Comm[175..179]: 5*)
		FOReturnDelay : REAL;
		FOPurgingDuration : REAL;
		FODSFlushingReserved2 : REAL;
		FODSFlushingReserved3 : REAL;
		FODSFlushingReserved4 : REAL;
	END_STRUCT;
	CommonReservedCat3_typ : 	STRUCT
		CommReserved180 : REAL;
		CommReserved181 : REAL;
		CommReserved182 : REAL;
		CommReserved183 : REAL;
		CommReserved184 : REAL;
		CommReserved185 : REAL;
		CommReserved186 : REAL;
		CommReserved187 : REAL;
		CommReserved188 : REAL;
		CommReserved189 : REAL;
		CommReserved190 : REAL;
		CommReserved191 : REAL;
		CommReserved192 : REAL;
		CommReserved193 : REAL;
		CommReserved194 : REAL;
		CommReserved195 : REAL;
		CommReserved196 : REAL;
		CommReserved197 : REAL;
		CommReserved198 : REAL;
		CommReserved199 : REAL;
	END_STRUCT;
	FFpara_typ : 	STRUCT
		NumTableRow : REAL;
		HeatLossTemp : REAL;
	END_STRUCT;
	EngineLoad_typ : 	STRUCT
		EngineLoad0 : REAL;
		EngineLoad1 : REAL;
		EngineLoad2 : REAL;
		EngineLoad3 : REAL;
		EngineLoad4 : REAL;
		EngineLoad5 : REAL;
		EngineLoad6 : REAL;
		EngineLoad7 : REAL;
		EngineLoad8 : REAL;
		EngineLoad9 : REAL;
		EngineLoad10 : REAL;
		EngineLoad11 : REAL;
	END_STRUCT;
	ExhFlowrate_typ : 	STRUCT
		ExhFlowrate0 : REAL;
		ExhFlowrate1 : REAL;
		ExhFlowrate2 : REAL;
		ExhFlowrate3 : REAL;
		ExhFlowrate4 : REAL;
		ExhFlowrate5 : REAL;
		ExhFlowrate6 : REAL;
		ExhFlowrate7 : REAL;
		ExhFlowrate8 : REAL;
		ExhFlowrate9 : REAL;
		ExhFlowrate10 : REAL;
		ExhFlowrate11 : REAL;
	END_STRUCT;
	HUInletRefTemp_typ : 	STRUCT
		HUInletRefTemp0 : REAL;
		HUInletRefTemp1 : REAL;
		HUInletRefTemp2 : REAL;
		HUInletRefTemp3 : REAL;
		HUInletRefTemp4 : REAL;
		HUInletRefTemp5 : REAL;
		HUInletRefTemp6 : REAL;
		HUInletRefTemp7 : REAL;
		HUInletRefTemp8 : REAL;
		HUInletRefTemp9 : REAL;
		HUInletRefTemp10 : REAL;
		HUInletRefTemp11 : REAL;
	END_STRUCT;
	CorrectionFactor_typ : 	STRUCT
		CorrectionFactor0 : REAL;
		CorrectionFactor1 : REAL;
		CorrectionFactor2 : REAL;
		CorrectionFactor3 : REAL;
		CorrectionFactor4 : REAL;
		CorrectionFactor5 : REAL;
		CorrectionFactor6 : REAL;
		CorrectionFactor7 : REAL;
		CorrectionFactor8 : REAL;
		CorrectionFactor9 : REAL;
		CorrectionFactor10 : REAL;
		CorrectionFactor11 : REAL;
	END_STRUCT;
	MOCSTempPgain_typ : 	STRUCT
		MOCSTempPgain0 : REAL;
		MOCSTempPgain1 : REAL;
		MOCSTempPgain2 : REAL;
		MOCSTempPgain3 : REAL;
		MOCSTempPgain4 : REAL;
		MOCSTempPgain5 : REAL;
		MOCSTempPgain6 : REAL;
		MOCSTempPgain7 : REAL;
		MOCSTempPgain8 : REAL;
		MOCSTempPgain9 : REAL;
		MOCSTempPgain10 : REAL;
		MOCSTempPgain11 : REAL;
	END_STRUCT;
	APIDgain_typ : 	STRUCT
		MOCSTempIgain : REAL;
		MOCSTempDgain : REAL;
		MOCSTempNoiseSup : REAL;
		QFOPgain : REAL;
		QFOIgain : REAL;
		QFODgain : REAL;
		QFONoiseSup : REAL;
		FODSFeedbackReserved19 : REAL;
		FODSFeedbackReserved20 : REAL;
		FODSFeedbackReserved21 : REAL;
		FODSFeedbackReserved22 : REAL;
		FODSFeedbackReserved23 : REAL;
		FODSFeedbackReserved24 : REAL;
	END_STRUCT;
	IndivReservedCat3_typ : 	STRUCT
		IndivReserved75 : REAL;
		IndivReserved76 : REAL;
		IndivReserved77 : REAL;
		IndivReserved78 : REAL;
		IndivReserved79 : REAL;
		IndivReserved80 : REAL;
		IndivReserved81 : REAL;
		IndivReserved82 : REAL;
		IndivReserved83 : REAL;
		IndivReserved84 : REAL;
		IndivReserved85 : REAL;
		IndivReserved86 : REAL;
		IndivReserved87 : REAL;
		IndivReserved88 : REAL;
		IndivReserved89 : REAL;
		IndivReserved90 : REAL;
		IndivReserved91 : REAL;
		IndivReserved92 : REAL;
		IndivReserved93 : REAL;
		IndivReserved94 : REAL;
		IndivReserved95 : REAL;
		IndivReserved96 : REAL;
		IndivReserved97 : REAL;
		IndivReserved98 : REAL;
		IndivReserved99 : REAL;
	END_STRUCT;
END_TYPE
```


### Program Logical/Package/COSMO_SET (IEC)

#### Variables.var
```iecst
VAR
	idx : USINT;
END_VAR
```

#### Main.st
```iecst
PROGRAM _INIT
	(* Insert code here *)
	OpcUA_cmd;
	OpcUA_modifier;
	OpcUA_mon;
	OpcUA_set_1[0] := 0;
	//OpcUA_set_15[0] := 0;
	//OpcUA_set_30[0] := 0;
END_PROGRAM

PROGRAM _CYCLIC
	(* Insert code here *)

	OpcUA_mon[0] := 100;
	IF OpcUA_set_1[0] = 1 THEN
		FOR idx := 1 TO 10 DO
			OpcUA_mon[10+idx] := OpcUA_set_1[idx];
		END_FOR;
			OpcUA_set_1[0] := 0;
	END_IF;
END_PROGRAM

PROGRAM _EXIT
	(* Insert code here *)

END_PROGRAM
```

### MAT_IO.var
```iecst
VAR
	X20IOSim : X20IOMat_typ;
	X20IOMat : X20IOMat_typ;
END_VAR
```

### MAT_IO.typ
```iecst
TYPE
	X20IOMat_typ : 	STRUCT
		CommModule : Common_MAT_typ;
		IndivModule : ARRAY[0..7]OF Indiv_MAT_typ;
	END_STRUCT;
	Common_MAT_typ : 	STRUCT
		DIF371 : DIF371_MAT_typ;
		DOF322 : DOF322_MAT_typ;
		AI8321 : AI8321_MAT_typ;
	END_STRUCT;
	Indiv_MAT_typ : 	STRUCT
		DIF371 : DIF371_MAT_typ;
		DOF322 : DOF322_MAT_typ;
		AI8321 : ARRAY[0..2]OF AI8321_MAT_typ;
		AO4622 : AO4622_MAT_typ;
	END_STRUCT;
	DIF371_MAT_typ : 	STRUCT
		Value : ARRAY[0..15]OF BOOL;
	END_STRUCT;
	DOF322_MAT_typ : 	STRUCT
		Value : ARRAY[0..15]OF BOOL;
	END_STRUCT;
	AI8321_MAT_typ : 	STRUCT
		Value : ARRAY[0..7]OF REAL;
	END_STRUCT;
	AO4622_MAT_typ : 	STRUCT
		Value : ARRAY[0..3]OF REAL;
	END_STRUCT;
END_TYPE
```

### Program Logical/IODefinitions/IODiver (IEC)

#### IODiver.st - Init, cyclic, exit code
```iecst
PROGRAM _INIT
	(* Insert code here *)
	StructTest;
	IF_MON;
	IF_PARA;		// Shutdown
	IF_PARA_Comm;	// Shutdown
	IF_PARA_CSys;	// Generated
	IF_PARA_CFlag;	// Generated
	IF_PARA_CMain;	// Generated
	IF_PARA_CFODS;	// Generated
	IF_PARA_CReserved;	// Generated
	IF_PARA_No1FF;
	IF_PARA_No1FB;
	IF_PARA_No1Reserved;
	IF_PARA_No2FF;
	IF_PARA_No2FB;
	IF_PARA_No2Reserved;
	IF_PARA_No3FF;
	IF_PARA_No3FB;
	IF_PARA_No3Reserved;
	IF_PARA_No4FF;
	IF_PARA_No4FB;
	IF_PARA_No4Reserved;
	IF_PARA_No5FF;
	IF_PARA_No5FB;
	IF_PARA_No5Reserved;
	IF_PARA_No6FF;
	IF_PARA_No6FB;
	IF_PARA_No6Reserved;
	IF_PARA_No7FF;
	IF_PARA_No7FB;
	IF_PARA_No7Reserved;
	IF_PARA_No8FF;
	IF_PARA_No8FB;
	IF_PARA_No8Reserved;
END_PROGRAM

PROGRAM _CYCLIC
	(* Insert code here *)
//	StructTest;
//	IF_MON;
END_PROGRAM

PROGRAM _EXIT
	(* Insert code here *)

END_PROGRAM
```

### IO.var
```iecst
VAR
	StructTest : StructTest_typ;
END_VAR
```

### IO.typ
```iecst
TYPE
	StructTest_typ : 	STRUCT
		R0 : REAL;
		R1 : REAL;
		R2 : REAL;
	END_STRUCT;
END_TYPE
```

### Program Logical/CtrlLogic

#### MOCS_AS_Gen.h
```c
/********************************************************************
 * COPYRIGHT -- B&R Industrial Automation GmbH
 ********************************************************************
 * Program: MOCS_AS_Gen
 * File: MOCS_AS_Gen.h
 * Author: HHI
 * Last modified by: HHI
 * Created: Mon Nov 17 13:23:17 2025
 * Last modified: Fri Nov 21 16:29:48 2025
 * Model Version: 5.11
 * Description:
 * modified Comment:
 ********************************************************************
 * Header for program MOCS_AS_Gen
 ********************************************************************
 * Generated with B&R Automation Studio Target for Simulink V7.1.1
 * (ERT based)
 ********************************************************************/

#ifndef MOCS_AS_Gen_h_
#define MOCS_AS_Gen_h_
#ifndef MOCS_AS_Gen_COMMON_INCLUDES_
#define MOCS_AS_Gen_COMMON_INCLUDES_
#include "rtwtypes.h"
#include "rtw_continuous.h"
#include "rtw_solver.h"
#endif                                 /* MOCS_AS_Gen_COMMON_INCLUDES_ */

#include <bur/plctypes.h>

#ifdef _DEFAULT_INCLUDES
 #include <AsDefault.h>
#endif

#ifndef AST_ROUND
#define AST_ROUND(x) ((x)>=0?(long long)((x)+0.5):(long long)((x)-0.5))
#endif

#include "MOCS_AS_Gen_types.h"

/* Macros for accessing real-time model data structure */
#ifndef rtmGetErrorStatus
#define rtmGetErrorStatus(rtm)         ((rtm)->errorStatus)
#endif

#ifndef rtmSetErrorStatus
#define rtmSetErrorStatus(rtm, val)    ((rtm)->errorStatus = (val))
#endif

#ifndef MIN
#define MIN(a,b)                       ((a) < (b) ? (a) : (b))
#endif

#ifndef MAX
#define MAX(a,b)                       ((a) > (b) ? (a) : (b))
#endif

#ifndef AST_ROUND
#define AST_ROUND(x)                   ((x)>=0?(long long)((x)+0.5):(long long)((x)-0.5))
#endif

/* Block signals (default storage) */
typedef struct {
  CMDO_typ System;                     /* '<Root>/Ext Struct In2' */
  CMDO_typ BusConversion_InsertedFor_ExtSt;
} BlockIO_MOCS_AS_Gen;

/* Real-time Model Data Structure */
struct tag_RTM_MOCS_AS_Gen {
  const char_T * volatile errorStatus;
};

/* Block signals (default storage) */
extern BlockIO_MOCS_AS_Gen MOCS_AS_Gen_B;

/* Model entry point functions */
extern void MOCS_AS_Gen_initialize(void);
extern void MOCS_AS_Gen_output(void);
extern void MOCS_AS_Gen_update(void);
extern void MOCS_AS_Gen_terminate(void);

/* Real-time Model object */
extern RT_MODEL_MOCS_AS_Gen *const MOCS_AS_Gen_M;

/*-
 * The generated code includes comments that allow you to trace directly
 * back to the appropriate location in the model.  The basic format
 * is <system>/block_name, where system is the system number (uniquely
 * assigned by Simulink) and block_name is the name of the block.
 *
 * Use the MATLAB hilite_system command to trace the generated code back
 * to the model.  For example,
 *
 * hilite_system('<S3>')    - opens system 3
 * hilite_system('<S3>/Kp') - opens and selects block Kp which resides in S3
 *
 * Here is the system hierarchy for this model
 *
 * '<Root>' : 'MOCS_AS_Gen'
 */
#endif                                 /* MOCS_AS_Gen_h_ */
```

#### MOCS_AS_Gen_types.h
```c
/********************************************************************
 * COPYRIGHT -- B&R Industrial Automation GmbH
 ********************************************************************
 * Program: MOCS_AS_Gen
 * File: MOCS_AS_Gen_types.h
 * Author: HHI
 * Last modified by: HHI
 * Created: Mon Nov 17 13:23:17 2025
 * Last modified: Fri Nov 21 16:29:48 2025
 * Model Version: 5.11
 * Description:
 * modified Comment:
 ********************************************************************
 * Header for program MOCS_AS_Gen
 ********************************************************************
 * Generated with B&R Automation Studio Target for Simulink V7.1.1
 * (ERT based)
 ********************************************************************/

#ifndef MOCS_AS_Gen_types_h_
#define MOCS_AS_Gen_types_h_
#include "rtwtypes.h"
#ifndef MIN
#define MIN(a,b)                       ((a) < (b) ? (a) : (b))
#endif

#ifndef MAX
#define MAX(a,b)                       ((a) > (b) ? (a) : (b))
#endif

#ifndef AST_ROUND
#define AST_ROUND(x)                   ((x)>=0?(long long)((x)+0.5):(long long)((x)-0.5))
#endif

/* Forward declaration for rtModel */
typedef struct tag_RTM_MOCS_AS_Gen RT_MODEL_MOCS_AS_Gen;

#endif                                 /* MOCS_AS_Gen_types_h_ */
```

#### rtwtypes.h
```c
/********************************************************************
 * COPYRIGHT -- B&R Industrial Automation GmbH
 ********************************************************************
 * Program: MOCS_AS_Gen
 * File: rtwtypes.h
 * Author: HHI
 * Last modified by: HHI
 * Created: Mon Nov 17 13:23:17 2025
 * Last modified: Fri Nov 21 16:29:48 2025
 * Model Version: 5.11
 * Description:
 * modified Comment:
 ********************************************************************
 * Header for program MOCS_AS_Gen
 ********************************************************************
 * Generated with B&R Automation Studio Target for Simulink V7.1.1
 * (ERT based)
 ********************************************************************/

#ifndef RTWTYPES_H
#define RTWTYPES_H

/* Logical type definitions */
#if (!defined(__cplusplus))
#ifndef false
#define false                          (0U)
#endif

#ifndef true
#define true                           (1U)
#endif
#endif

/*=======================================================================*
 * Target hardware information
 *   Device type: Intel->x86/Pentium
 *   Number of bits:     char:   8    short:   16    long:  32
 *                       long:  32
 *                       native word size:  32
 *   Byte ordering: LittleEndian
 *   Signed integer division rounds to: Zero
 *   Shift right on a signed integer as arithmetic shift: on
 *=======================================================================*/

/*=======================================================================*
 * Fixed width word size data types:                                     *
 *   int8_T, int16_T, int32_T     - signed 8, 16, or 32 bit integers     *
 *   uint8_T, uint16_T, uint32_T  - unsigned 8, 16, or 32 bit integers   *
 *   real32_T, real64_T           - 32 and 64 bit floating point numbers *
 *=======================================================================*/
typedef signed char int8_T;
typedef unsigned char uint8_T;
typedef short int16_T;
typedef unsigned short uint16_T;
typedef long int32_T;
typedef unsigned long uint32_T;
typedef float real32_T;
typedef double real64_T;

/*===========================================================================*
 * Generic type definitions: boolean_T, char_T, byte_T, int_T, uint_T,       *
 *                           real_T, time_T, ulong_T.                        *
 *===========================================================================*/
typedef double real_T;
typedef double time_T;
typedef unsigned char boolean_T;
typedef long int_T;
typedef unsigned long uint_T;
typedef unsigned long ulong_T;
typedef char char_T;
typedef unsigned char uchar_T;
typedef char_T byte_T;

/*===========================================================================*
 * Complex number type definitions                                           *
 *===========================================================================*/
#define CREAL_T

typedef struct {
  real32_T re;
  real32_T im;
} creal32_T;

typedef struct {
  real64_T re;
  real64_T im;
} creal64_T;

typedef struct {
  real_T re;
  real_T im;
} creal_T;

#define CINT8_T

typedef struct {
  int8_T re;
  int8_T im;
} cint8_T;

#define CUINT8_T

typedef struct {
  uint8_T re;
  uint8_T im;
} cuint8_T;

#define CINT16_T

typedef struct {
  int16_T re;
  int16_T im;
} cint16_T;

#define CUINT16_T

typedef struct {
  uint16_T re;
  uint16_T im;
} cuint16_T;

#define CINT32_T

typedef struct {
  int32_T re;
  int32_T im;
} cint32_T;

#define CUINT32_T

typedef struct {
  uint32_T re;
  uint32_T im;
} cuint32_T;

/*=======================================================================*
 * Min and Max:                                                          *
 *   int8_T, int16_T, int32_T     - signed 8, 16, or 32 bit integers     *
 *   uint8_T, uint16_T, uint32_T  - unsigned 8, 16, or 32 bit integers   *
 *=======================================================================*/
#define MAX_int8_T                     ((int8_T)(127))
#define MIN_int8_T                     ((int8_T)(-128))
#define MAX_uint8_T                    ((uint8_T)(255U))
#define MAX_int16_T                    ((int16_T)(32767))
#define MIN_int16_T                    ((int16_T)(-32768))
#define MAX_uint16_T                   ((uint16_T)(65535U))
#define MAX_int32_T                    ((int32_T)(2147483647))
#define MIN_int32_T                    ((int32_T)(-2147483647-1))
#define MAX_uint32_T                   ((uint32_T)(0xFFFFFFFFU))

/* Block D-Work pointer type */
typedef void * pointer_T;

#endif                                 /* RTWTYPES_H */

#ifndef MIN
#define MIN(a,b)                       ((a) < (b) ? (a) : (b))
#endif

#ifndef MAX
#define MAX(a,b)                       ((a) > (b) ? (a) : (b))
#endif

#ifndef AST_ROUND
#define AST_ROUND(x)                   ((x)>=0?(long long)((x)+0.5):(long long)((x)-0.5))
#endif
```

#### CtrlLogic.c
```c
/********************************************************************
 * COPYRIGHT -- B&R Industrial Automation GmbH
 ********************************************************************
 * Program: MOCS_AS_Gen
 * File: CtrlLogic.c
 * Author: HHI
 * Last modified by: HHI
 * Created: Mon Nov 17 13:23:17 2025
 * Last modified: Fri Nov 21 16:29:48 2025
 * Model Version: 5.11
 * Description:
 * modified Comment:
 ********************************************************************
 * Implementation of program MOCS_AS_Gen
 ********************************************************************
 * Generated with B&R Automation Studio Target for Simulink V7.1.1
 * (ERT based)
 ********************************************************************/

#define _ASMATH_
#define ASMATH_
#define _ASMATH_H
#define ASMATH_H
#define _ASMATH_H_
#define ASMATH_H_
#define _ASSTRING_
#define ASSTRING_
#define _ASSTRING_H
#define ASSTRING_H
#define _ASSTRING_H_
#define ASSTRING_H_
#include <bur/plctypes.h>
#ifdef _DEFAULT_INCLUDES
#include <AsDefault.h>
#endif

#include "MOCS_AS_Gen.h"
#include "rtwtypes.h"

/*  Defines */

/*  Data Types */

/**************************** GLOBAL DATA *************************************/
/*  Definitions */

/*  Declarations  */

/***************************** FILE SCOPE DATA ********************************/

/*************************** FUNCTIONS ****************************************/
#ifdef __cplusplus

unsigned long bur_heap_size = 6553500;

#endif

  void _INIT mainINIT(void)
{

    UDINT st_ident;
  RTInfo_typ rt_info;
  rt_info.enable = 1;
  RTInfo(&rt_info);
  if (rt_info.cycle_time != 100000) {
    /* cycle time does not match Simulink fixed-step size */
    ST_ident("CtrlLogic", 0, &st_ident);
    ST_tmp_suspend(st_ident);
    ERR_warning(33310, 0);
  }

  /* initialize model */
  MOCS_AS_Gen_initialize();

} void _CYCLIC mainCYCLIC(void)
{
  /* call model step function */
  MOCS_AS_Gen_output();

  MOCS_AS_Gen_update();

} void _EXIT mainEXIT(void)
{
  /* terminate model */
  MOCS_AS_Gen_terminate();

} /*****************************************************************************
     Task sample time: 0.099999999999999992s
   *****************************************************************************/
/*****************************************************************************
   B&R Automation Studio Target for Simulink Version: V7.1.1 (19-Sep-2025)
 *****************************************************************************/

/*======================== TOOL VERSION INFORMATION ==========================*
 * MATLAB 24.2 (R2024b)21-Jun-2024                                            *
 * Simulink 24.2 (R2024b)21-Jun-2024                                          *
 * Simulink Coder 24.2 (R2024b)21-Jun-2024                                    *
 * Embedded Coder 24.2 (R2024b)21-Jun-2024                                    *
 * Stateflow 24.2 (R2024b)21-Jun-2024                                         *
 * Fixed-Point Designer 24.2 (R2024b)21-Jun-2024                              *
 *============================================================================*/

/*======================= LICENSE IN USE INFORMATION =========================*
 * matlab                                                                     *
 * matlab_coder                                                               *
 * real-time_workshop                                                         *
 * rtw_embedded_coder                                                         *
 * simulink                                                                   *
 *============================================================================*/
```

#### global.txt
```
VAR
        Test_out : CMDO_typ; (**)
        Test_In : CMDO_typ; (**)
END_VAR
```

#### MOCS_AS_Gen_data.c
```c
/********************************************************************
 * COPYRIGHT -- B&R Industrial Automation GmbH
 ********************************************************************
 * Program: MOCS_AS_Gen
 * File: MOCS_AS_Gen_data.c
 * Author: HHI
 * Last modified by: HHI
 * Created: Mon Nov 17 13:23:17 2025
 * Last modified: Fri Nov 21 15:11:31 2025
 * Model Version: 5.5
 * Description:
 * modified Comment:
 ********************************************************************
 * Data for program MOCS_AS_Gen
 ********************************************************************
 * Generated with B&R Automation Studio Target for Simulink V7.1.1
 * (ERT based)
 ********************************************************************/

#include "MOCS_AS_Gen.h"

/*  GLOBAL DATA DEFINITIONS */

/* Block parameters (default storage) */
Parameters_MOCS_AS_Gen MOCS_AS_Gen_P = {
  /* Expression: 1
   * Referenced by: '<Root>/Constant'
   */
  1.0,

  /* Expression: 1
   * Referenced by: '<Root>/Constant1'
   */
  1.0,

  /* Expression: 1
   * Referenced by: '<Root>/Constant2'
   */
  1.0
};
```

### Package Logical/MATLAB_includes - Default includes for B&R Automation Studio Target for Simulink

### Package Logical/MATLAB_includes/R2024b - Default includes for MATLAB R2024b

### MAT_IF.var
```iecst
(*---MATLAB Input---*)
VAR
	IF_PARA : Para_typ; (*MAT IN*)
	IF_ALARM : Alarm_typ; (*MAT IN*)
END_VAR
```

### MAT_AL.typ
```iecst
(*---Category1---*)

TYPE
	Alarm_typ :	STRUCT
		Comm : CommAlarm_typ;
		No1 : IndivAlarm_typ;
		No2 : IndivAlarm_typ;
		No3 : IndivAlarm_typ;
		No4 : IndivAlarm_typ;
		No5 : IndivAlarm_typ;
		No6 : IndivAlarm_typ;
		No7 : IndivAlarm_typ;
		No8 : IndivAlarm_typ;
	END_STRUCT;
END_TYPE

(*---Category2---*)

TYPE
	CommAlarm_typ :	STRUCT
		CHD : CHD_typ;
		CUD : CUD_typ;
	END_STRUCT;
	IndivAlarm_typ :	STRUCT
		IHD : IHD_typ;
		IUD : IUD_typ;
	END_STRUCT;
END_TYPE

(*---Category3---*)

TYPE
	CHD_typ :	STRUCT
		CommonAI1ModuleFault : BOOL;
		CommonDI1ModuleFault : BOOL;
		CommonDO1ModuleFault : BOOL;
		FOpumpAutomode_HA : DIAlarm_typ;
		AlarmReset_HR : DIAlarm_typ;
		LCpowerFail_LF : DIAlarm_typ;
		InternalpowerFail_LF : DIAlarm_typ;
		ExternalpowerFail_LF : DIAlarm_typ;
		FanpowerFail_LF : DIAlarm_typ;
		ESDcircuitpowerFail_LF : DIAlarm_typ;
		No1FOpumpRemote_HR : DIAlarm_typ;
		No1FOpumpAbnormal_LA : DIAlarm_typ;
		No1FOpumpRunning_HR : DIAlarm_typ;
		No2FOpumpRemote_HR : DIAlarm_typ;
		No2FOpumpAbnormal_LA : DIAlarm_typ;
		No2FOpumpRunning_HR : DIAlarm_typ;
		CDI1CH14Reserved_HR : DIAlarm_typ;
		CDI1CH15Reserved_HR : DIAlarm_typ;
		CDI1CH16Reserved_HR : DIAlarm_typ;
		FOSupplyInletPress : AIAlarm_typ;
		FOSupplyOutletPress : AIAlarm_typ;
		CAI1CH3Reserved : AIAlarm_typ;
		CAI1CH4Reserved : AIAlarm_typ;
		CAI1CH5Reserved : AIAlarm_typ;
		CAI1CH6Reserved : AIAlarm_typ;
		CAI1CH7Reserved : AIAlarm_typ;
		CAI1CH8Reserved : AIAlarm_typ;
	END_STRUCT;
	CUD_typ :	STRUCT
		CommunicationFailwithHMI : BOOL;
		No1FOsupplypumpFail : BOOL;
		No2FOsupplypumpFail : BOOL;
	END_STRUCT;
	IHD_typ :	STRUCT
		AI1ModuleFault : BOOL;
		AI2ModuleFault : BOOL;
		AI3ModuleFault : BOOL;
		AO1ModuleFault : BOOL;
		DI1ModuleFault : BOOL;
		DO1ModuleFault : BOOL;
		LowSulfurfuelsupplied_H0 : DIAlarm_typ;
		MOCSRemoteLocal_HR : DIAlarm_typ;
		MOCSEmcystopFpanel_LE : DIAlarm_typ;
		MOCSEmcystopFECR_LE : DIAlarm_typ;
		MOCSEmcystopFBridge_LE : DIAlarm_typ;
		MOCSStart_HS : DIAlarm_typ;
		MOCSPreparation_HP : DIAlarm_typ;
		MOCSStop_HS : DIAlarm_typ;
		RSVFeedback_HO : DIAlarm_typ;
		RSVFeedback_HC : DIAlarm_typ;
		RBVFeedback_HO : DIAlarm_typ;
		RBVFeedback_HC : DIAlarm_typ;
		FODosFOInletTemp_L  : DIAlarm_typ;
		SCRValveFeedback_HO : DIAlarm_typ;
		SCRValveFeedback_HC : DIAlarm_typ;
		DI1CH16Reserved_HC : DIAlarm_typ;
		MixerInletTemp : AIAlarm_typ;
		ChamberInletTemp : AIAlarm_typ;
		ChamberMiddleTemp : AIAlarm_typ;
		ChamberOutletTemp : AIAlarm_typ;
		ChamberDiffPress : AIAlarm_typ;
		VnSAirInletPress : AIAlarm_typ;
		AI1CH7Reserved : AIAlarm_typ;
		AI1CH8Reserved : AIAlarm_typ;
		RBVPDT : AIAlarm_typ;
		RTVPDT : AIAlarm_typ;
		RTVFeedback : AIAlarm_typ;
		AI2CH4Reserved : AIAlarm_typ;
		AI2CH5Reserved : AIAlarm_typ;
		AI2CH6Reserved : AIAlarm_typ;
		AI2CH7Reserved : AIAlarm_typ;
		AI2CH8Reserved : AIAlarm_typ;
		FODosAirInletPress : AIAlarm_typ;
		FODosAirOutletPress : AIAlarm_typ;
		FODosFOInletPress : AIAlarm_typ;
		FODosFOMiddlePress : AIAlarm_typ;
		FODosFOFlowrateFeedback : AIAlarm_typ;
		FODosFOOutletPress : AIAlarm_typ;
		AI3CH7Reserved : AIAlarm_typ;
		AI3CH8Reserved : AIAlarm_typ;
	END_STRUCT;
	IUD_typ :	STRUCT
		CommunicationFailwithAMS : BOOL;
		EGSuddenDieselTransfer : BOOL;
		EGstoppedduringgas : BOOL;
		MSSNormalFail : BOOL;
		TMBTimeout : BOOL;
		RemoteStopWhileTMB : BOOL;
		MOCSNotReady : BOOL;
		RSVFail : BOOL;
		RSVFeedbackSF : BOOL;
		RBVFail : BOOL;
		RBVFeedbackSF : BOOL;
		SCRValveFail : BOOL;
		SCRValveFeedbackSF : BOOL;
		RTVFail : BOOL;
		RTVDev : BOOL;
		DosingFOFlowDev : BOOL;
		DosingFOFlowDevTimeout : BOOL;
		DosingFOLimitSatTimeout : BOOL;
		RTVPDTSFMOCSNotready : BOOL;
	END_STRUCT;
END_TYPE

(*---Category3---*)

TYPE
	AIAlarm_typ :	STRUCT
		SF : BOOL;
		LL : BOOL;
		LO : BOOL;
		HO : BOOL;
		HH : BOOL;
	END_STRUCT;
	DIAlarm_typ :	STRUCT
		DH : BOOL;
		DL : BOOL;
	END_STRUCT;
END_TYPE
```

### MAT_IO.var
```iecst
VAR
	IF_MATIN_IO : IO_typ;
	IF_MATOUT_IO : IndivIO_typ;
END_VAR
```

### MAT_IO.typ
```iecst
(*---Category1---*)

TYPE
	IO_typ :	STRUCT
		Comm : CommIO_typ;
		No1 : IndivIO_typ;
		No2 : IndivIO_typ;
		No3 : IndivIO_typ;
		No4 : IndivIO_typ;
		No5 : IndivIO_typ;
		No6 : IndivIO_typ;
		No7 : IndivIO_typ;
		No8 : IndivIO_typ;
	END_STRUCT;
END_TYPE

(*---Category2---*)

TYPE
	CommIO_typ :	STRUCT
		CAI : CAI_typ;
		CDI : CDI_typ;
		CDO : CDO_typ;
	END_STRUCT;
	IndivIO_typ :	STRUCT
		IAI : IAI_typ;
		IDI : IDI_typ;
		IAO : IAO_typ;
		IDO : IDO_typ;
	END_STRUCT;
END_TYPE

(*---Category3_Comm---*)

TYPE
	CAI_typ :	STRUCT
		FOSupplyInletPress : REAL;
		FOSupplyOutletPress : REAL;
		CAI1Reserved3 : REAL;
		CAI1Reserved4 : REAL;
		CAI1Reserved5 : REAL;
		CAI1Reserved6 : REAL;
		CAI1Reserved7 : REAL;
		CAI1Reserved8 : REAL;
	END_STRUCT;
	CDI_typ :	STRUCT
		FOSupplypumpAutomode : BOOL;
		AlarmReset : BOOL;
		PLCpowerFail_Reserved : BOOL;
		InternalpowerFail : BOOL;
		ExternalpowerFail : BOOL;
		FanpowerFail : BOOL;
		ESDcircuitpowerFail : BOOL;
		No1FOSupplypumpRemote : BOOL;
		No1FOSupplypumpAbnormal : BOOL;
		No1FOSupplypumpRunning : BOOL;
		No2FOSupplypumpRemote : BOOL;
		No2FOSupplypumpAbnormal : BOOL;
		No2FOSupplypumpRunning : BOOL;
		fromYardFOSupplypumpRunning : BOOL;
		CDI1Reserved15 : BOOL;
		CDI1Reserved16 : BOOL;
	END_STRUCT;
	CDO_typ :	STRUCT
		MOCSCommonAlarm : BOOL;
		MOCSCommonAlarmLamp : BOOL;
		MOCSCommonAlarmBuzzer : BOOL;
		No1FOSupplypumpRunCommand : BOOL;
		No2FOSupplypumpRunCommand : BOOL;
		toYardFOSupplypumpRunRequest : BOOL;
		toYardFOSupplypumpFail : BOOL;
		CDO1Reserved8 : BOOL;
		CDO1Reserved9 : BOOL;
		CDO1Reserved10 : BOOL;
		CDO1Reserved11 : BOOL;
		CDO1Reserved12 : BOOL;
		CDO1Reserved13 : BOOL;
		CDO1Reserved14 : BOOL;
		CDO1Reserved15 : BOOL;
		CDO1Reserved16 : BOOL;
	END_STRUCT;
END_TYPE

(*---Category3_Indiv---*)

TYPE
	IAI_typ :	STRUCT
		MixerInletTemp : REAL;
		ChamberInletTemp : REAL;
		ChamberMiddleTemp : REAL;
		ChamberOutletTemp : REAL;
		ChamberDiffPress : REAL;
		VentingSealingAirInletPress : REAL;
		IAI1Reserved7 : REAL;
		IAI1Reserved8 : REAL;
		RBVPDT : REAL;
		RTVPDT : REAL;
		RTVFeedback : REAL;
		IAI2Reserved4 : REAL;
		IAI2Reserved5 : REAL;
		IAI2Reserved6 : REAL;
		IAI2Reserved7 : REAL;
		IAI2Reserved8 : REAL;
		FODAtomizingAirInletPress : REAL;
		FODAtomizingAirOutletPress : REAL;
		FODFuelOilInletPress : REAL;
		FODFuelOilMiddlePress : REAL;
		FODFuelOilFlowrate_Feedback : REAL;
		FODFuelOilOutletPress : REAL;
		IAI3Reserved7 : REAL;
		IAI3Reserved8 : REAL;
	END_STRUCT;
	IDI_typ :	STRUCT
		GELowSulfurfuelsupplied : BOOL;
		MOCSRemoteLocal : BOOL;
		MOCSEmcystopFrompanel : BOOL;
		MOCSEmcystopFromECR : BOOL;
		MOCSEmcystopFromBridge : BOOL;
		MOCSStart : BOOL;
		MOCSPreparation : BOOL;
		MOCSStop : BOOL;
		RSVFeedback_Open : BOOL;
		RSVFeedback_Closed : BOOL;
		RBVFeedback_Open : BOOL;
		RBVFeedback_Closed : BOOL;
		FODFuelOilInletTemp : BOOL;
		SCRValveFeedback_Open : BOOL;
		SCRValveFeedback_Close : BOOL;
		IDI1Reserved16 : BOOL;
	END_STRUCT;
	IAO_typ :	STRUCT
		FODFuelOilControlVV_Setpoint : REAL;
		RTVSetpoint : REAL;
		IAO1Reserved3 : REAL;
		IAO1Reserved4 : REAL;
	END_STRUCT;
	IDO_typ :	STRUCT
		MOCSReady : BOOL;
		AllFlowThroughMOCS : BOOL;
		MOCSActive : BOOL;
		MOCSFODsystemFlushRun : BOOL;
		FODAtomizingAirSolVV : BOOL;
		FODPurgingAirSolVV : BOOL;
		FODFuelOilInletSolVV : BOOL;
		FODFuelOilOutletSolVV : BOOL;
		FODFuelOilReturnSolVV : BOOL;
		RSVSetpoint : BOOL;
		RBVSetpoint : BOOL;
		VentingSealingSolVV : BOOL;
		SCRValveSetpoint : BOOL;
		IDO1Reserved14 : BOOL;
		IDO1Reserved15 : BOOL;
		IDO1Reserved16 : BOOL;
	END_STRUCT;
END_TYPE
```

### Program Logical/MATLAB_Interface/MAT_IO_test (IEC)

#### Main.st
```iecst
PROGRAM _INIT
	(* Insert code here *)
	IF_PARA;
	IF_MON;

END_PROGRAM

PROGRAM _CYCLIC
	(* Insert code here *)

END_PROGRAM

PROGRAM _EXIT
	(* Insert code here *)

END_PROGRAM
```

Listed in the project but not available here: Logical/Global.typ, Logical/MAT_IF.var, Logical/IODefinitions/IODiver/IODiver.typ, Logical/IODefinitions/IODiver/IODiver.var, Logical/MATLAB_includes/R2022b, Logical/MATLAB_includes/R2024b/MatlabDataArray.hpp, Logical/MATLAB_includes/R2024b/MatlabEngine.hpp, Logical/MATLAB_includes/R2024b/bio_sig.h, Logical/MATLAB_includes/R2024b/blas.h, Logical/MATLAB_includes/R2024b/blascompat32.h, Logical/MATLAB_includes/R2024b/cg_matrx.h, Logical/MATLAB_includes/R2024b/cg_sfun.h, Logical/MATLAB_includes/R2024b/cgxeooprt.h, Logical/MATLAB_includes/R2024b/cgxert.h, Logical/MATLAB_includes/R2024b/covrt.h, Logical/MATLAB_includes/R2024b/dt_info.h, Logical/MATLAB_includes/R2024b/emlrt.h, Logical/MATLAB_includes/R2024b/engine.h, Logical/MATLAB_includes/R2024b/ext_share.h, Logical/MATLAB_includes/R2024b/ext_svr.h, Logical/MATLAB_includes/R2024b/ext_svr_transport.h, Logical/MATLAB_includes/R2024b/ext_test.h, Logical/MATLAB_includes/R2024b/ext_types.h, Logical/MATLAB_includes/R2024b/ext_work.h, Logical/MATLAB_includes/R2024b/fintrf.h, Logical/MATLAB_includes/R2024b/fixedpoint.h, Logical/MATLAB_includes/R2024b/fixpoint_spec.h, Logical/MATLAB_includes/R2024b/i18n_c_api.h, Logical/MATLAB_includes/R2024b/io64.h, Logical/MATLAB_includes/R2024b/lapack.h, Logical/MATLAB_includes/R2024b/lapacke.h, Logical/MATLAB_includes/R2024b/lapacke_config.h, Logical/MATLAB_includes/R2024b/libmwjpegreader.h, Logical/MATLAB_includes/R2024b/libmwrgb2gray_tbb.h, Logical/MATLAB_includes/R2024b/libmwrgb2hsv_tbb.h, Logical/MATLAB_includes/R2024b/libmwslsa_engine.h, Logical/MATLAB_includes/R2024b/libmwslsa_sim.h, Logical/MATLAB_includes/R2024b/liveio.h, Logical/MATLAB_includes/R2024b/mat.h, Logical/MATLAB_includes/R2024b/matrix.h, Logical/MATLAB_includes/R2024b/mdl_info.h, Logical/MATLAB_includes/R2024b/mem_mgr.h, Logical/MATLAB_includes/R2024b/mex.h, Logical/MATLAB_includes/R2024b/mwmathutil.h, Logical/MATLAB_includes/R2024b/odesup.h, Logical/MATLAB_includes/R2024b/polygonBoolean.h, Logical/MATLAB_includes/R2024b/pt_info.h, Logical/MATLAB_includes/R2024b/rt_logging.h, Logical/MATLAB_includes/R2024b/rt_logging_mmi.h, Logical/MATLAB_includes/R2024b/rt_logging_simtarget.h, Logical/MATLAB_includes/R2024b/rt_math.h, Logical/MATLAB_includes/R2024b/rt_matrx.h, Logical/MATLAB_includes/R2024b/rt_mxclassid.h, Logical/MATLAB_includes/R2024b/rt_sim.h, Logical/MATLAB_includes/R2024b/rtiostream.h, Logical/MATLAB_includes/R2024b/rtmcmacros.h, Logical/MATLAB_includes/R2024b/rtmmacros.h, Logical/MATLAB_includes/R2024b/rtsplntypes.h, Logical/MATLAB_includes/R2024b/rtw_capi.h, Logical/MATLAB_includes/R2024b/rtw_capi_examples.h, Logical/MATLAB_includes/R2024b/rtw_continuous.h, Logical/MATLAB_includes/R2024b/rtw_extmode.h, Logical/MATLAB_includes/R2024b/rtw_linux.h, Logical/MATLAB_includes/R2024b/rtw_linux_mac.h, Logical/MATLAB_includes/R2024b/rtw_matlogging.h, Logical/MATLAB_includes/R2024b/rtw_matlogging_simtarget.h, Logical/MATLAB_includes/R2024b/rtw_modelmap.h, Logical/MATLAB_includes/R2024b/rtw_modelmap_logging.h, Logical/MATLAB_includes/R2024b/rtw_modelmap_simtarget.h, Logical/MATLAB_includes/R2024b/rtw_msvc_lshift.h, Logical/MATLAB_includes/R2024b/rtw_solver.h, Logical/MATLAB_includes/R2024b/rtw_storage.h, Logical/MATLAB_includes/R2024b/rtw_windows.h, Logical/MATLAB_includes/R2024b/sfcn_bridge.h, Logical/MATLAB_includes/R2024b/sfcn_loader_c_api.h, Logical/MATLAB_includes/R2024b/sfun_rtwcg.hpp, Logical/MATLAB_includes/R2024b/sigmapdef_sfcn.h, Logical/MATLAB_includes/R2024b/sigregdef.h, Logical/MATLAB_includes/R2024b/sigstream_rtw.h, Logical/MATLAB_includes/R2024b/simlogCIntrf.h, Logical/MATLAB_includes/R2024b/simstruc.h, Logical/MATLAB_includes/R2024b/simstruc_64_internal.h, Logical/MATLAB_includes/R2024b/simstruc_compcond.h, Logical/MATLAB_includes/R2024b/simstruc_debug.h, Logical/MATLAB_includes/R2024b/simstruc_def.h, Logical/MATLAB_includes/R2024b/simstruc_fwd.h, Logical/MATLAB_includes/R2024b/simstruc_genericfcn.h, Logical/MATLAB_includes/R2024b/simstruc_implement.h, Logical/MATLAB_includes/R2024b/simstruc_internal.h, Logical/MATLAB_includes/R2024b/simstruc_internal_types.h, Logical/MATLAB_includes/R2024b/simstruc_types.h, Logical/MATLAB_includes/R2024b/simulink.h, Logical/MATLAB_includes/R2024b/simulink2.h, Logical/MATLAB_includes/R2024b/simulink_solver_api.h, Logical/MATLAB_includes/R2024b/slImageTypes.h, Logical/MATLAB_includes/R2024b/sl_common_types_def.h, Logical/MATLAB_includes/R2024b/sl_datatype_access.h, Logical/MATLAB_includes/R2024b/sl_fileio_rtw.h, Logical/MATLAB_includes/R2024b/sl_fixpt.h, Logical/MATLAB_includes/R2024b/sl_prodhwdevicetype.h, Logical/MATLAB_includes/R2024b/sl_report_types.h, Logical/MATLAB_includes/R2024b/sl_sample_time_defs.h, Logical/MATLAB_includes/R2024b/sl_sfcn_st_api.h, Logical/MATLAB_includes/R2024b/sl_solver_rtw.h, Logical/MATLAB_includes/R2024b/sl_types_def.h, Logical/MATLAB_includes/R2024b/slccrt.h, Logical/MATLAB_includes/R2024b/slexec_block_runtime_service.h, Logical/MATLAB_includes/R2024b/slexec_parallel.h, Logical/MATLAB_includes/R2024b/slexec_simbridge.h, Logical/MATLAB_includes/R2024b/slexec_simstruct_bridge.h, Logical/MATLAB_includes/R2024b/slexec_ssExecutionInfo.h, Logical/MATLAB_includes/R2024b/slexec_vm_lookup_functions.h, Logical/MATLAB_includes/R2024b/slexec_vm_rt_functions.h, Logical/MATLAB_includes/R2024b/slexec_vm_simstruct_bridge.h, Logical/MATLAB_includes/R2024b/slexec_vm_zc_functions.h, Logical/MATLAB_includes/R2024b/slprocess.h, Logical/MATLAB_includes/R2024b/slsa_engine_exec.h, Logical/MATLAB_includes/R2024b/slsa_sim_engine.h, Logical/MATLAB_includes/R2024b/slsv_diagnostic_codegen_c_api.h, Logical/MATLAB_includes/R2024b/slsv_diagnostic_deployment_c_api.h, Logical/MATLAB_includes/R2024b/slsv_diagnostic_logger_type.h, Logical/MATLAB_includes/R2024b/slsv_mexhelper.h, Logical/MATLAB_includes/R2024b/solver_zc.h, Logical/MATLAB_includes/R2024b/sysran_types.h, Logical/MATLAB_includes/R2024b/tmwtypes.h, Logical/MATLAB_includes/R2024b/updown.h, Logical/MATLAB_includes/R2024b/updown_util.h, Logical/MATLAB_includes/R2024b/upsup_public.h, Logical/MATLAB_includes/R2024b/sf_runtime
